Omron CX-Programmer project NewProject (CX-Programmer 9.73)

# PLC projekat: CJ1M CPU11
I/O table (CPU CJ1M-CPU11): rack 0 slot 2 CJ1W-AD081-V1 "21"

## Global symbols (name address type ; comment)
0 CHANNEL  ; .
100 CHANNEL  ; Svetlo je upaljeno jos 10s
1.00 BOOL  ; Povecaj broj ljudi
C1 CHANNEL  ; Brojac ljudi koji su usli
D0 CHANNEL  ; Ulaz u sobu
D1.00 BOOL  ; Ljudi u prostoriji

## Program NewProgram1 (cyclic task 0)
Local symbols
Flag 200.00 BOOL  ; Nema nikoga u sobi
Flag2 200.01 BOOL  ; Za tajmer
Foto 2960.02 BOOL  ; Foto senzor
Noc 2960.04 BOOL  ; Kada je noc
PIR1 2960.01 BOOL  ; Senzor pokreta ulaza
PIR2 2960.03 BOOL  ; Senzor pokreta izlaza
Relej 2960.00 BOOL  ; Relej iskljucen
Svetlo 2961.00 BOOL  ; Lampa gori

### Section Section1

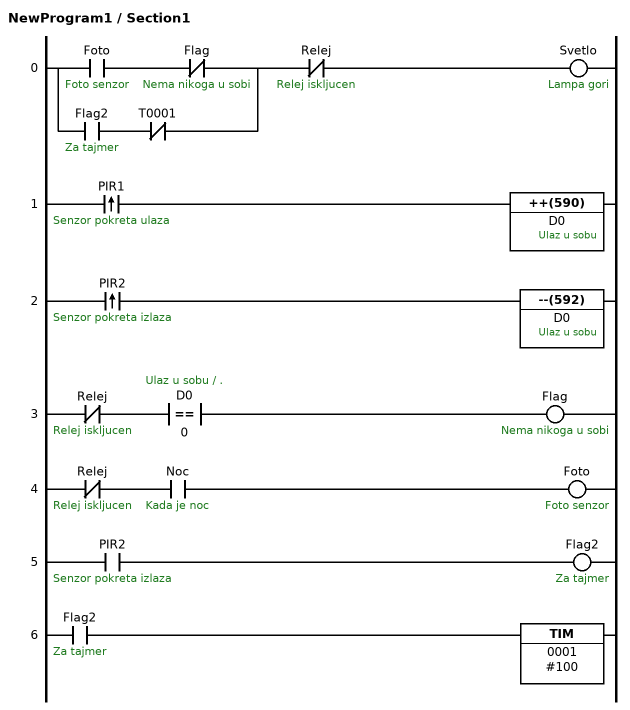
; rung 0
LD Foto  ; Foto senzor
ANDNOT Flag  ; Nema nikoga u sobi
LD Flag2  ; Za tajmer
ANDNOT T0001
ORLD
ANDNOT Relej  ; Relej iskljucen
OUT Svetlo  ; Lampa gori
; rung 1
@LD PIR1  ; Senzor pokreta ulaza
++(590) D0  ; Ulaz u sobu
; rung 2
@LD PIR2  ; Senzor pokreta izlaza
--(592) D0  ; Ulaz u sobu
; rung 3
LDNOT Relej  ; Relej iskljucen
AND=(300) D0 0  ; Ulaz u sobu, .
OUT Flag  ; Nema nikoga u sobi
; rung 4
LDNOT Relej  ; Relej iskljucen
AND Noc  ; Kada je noc
OUT Foto  ; Foto senzor
; rung 5
LD PIR2  ; Senzor pokreta izlaza
OUT Flag2  ; Za tajmer
; rung 6
LD Flag2  ; Za tajmer
TIM 0001 #100

### Section END
; rung 0
END(001)